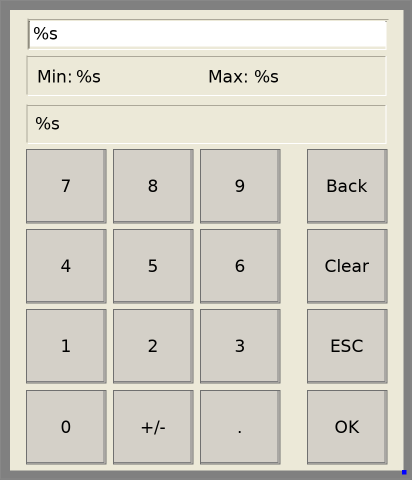
VISUALIZATION Custom_Numpad  // 412x480
VAR_INPUT
	stVariableValue : STRING;
	stMin : STRING;
	stMax : STRING;
	stTitle : STRING;
	flags : DWORD;
END_VAR
VAR
	bInit : BOOL;
	stMessage : STRING;
	stOutputValue : STRING;
END_VAR
    Rectangle (0,0 412x480)
    Rectangle (10,142 393x83)
    Rectangle (10,225 393x80)
    Rectangle (10,305 393x80)
    Rectangle (10,385 393x85)
    Button (307,390 80x74), "OK"
        OnMouseDown: CloseDialog Dialog=Custom_Numpad, Result=OK, NumpadKeypad=True, NumpadKeypadSet=True
    Button (307,309 80x74), "ESC"
        OnMouseDown: CloseDialog Dialog=Custom_Numpad, Result=Cancel, NumpadKeypad=True, NumpadKeypadSet=True
    Button (307,229 80x74), "Clear"
        OnMouseDown: execute {
            stVariableValue := '';
            stOutputValue := '';
            flags := flags AND 16#0008;
            flags := flags AND 16#0010;
        }
    Button (307,149 80x74), "Back"
        OnMouseDown: execute { VisuDlg_CheckedBack(stOutputValue, stVariableValue, bInit); }
    Button (200,390 80x74), "."
        OnMouseDown: execute { VisuDlg_CheckedAppend(stOutputValue, stVariableValue, bInit, (flags AND VisuElems.Visu_InputFlags.Password) = 1, '.'); }
    Button (113,390 80x74), "+/-"
        OnMouseDown: execute { VisuDlg_CheckedChangeSign(stOutputValue, stVariableValue, bInit, (flags AND VisuElems.Visu_InputFlags.Password) = 1); }
    Button (26,390 80x74), "0"
        OnMouseDown: execute { VisuDlg_CheckedAppend(stOutputValue, stVariableValue, bInit, (flags AND VisuElems.Visu_InputFlags.Password) = 1, '0'); }
    Button (26,309 80x74), "1"
        OnMouseDown: execute { VisuDlg_CheckedAppend(stOutputValue, stVariableValue, bInit, (flags AND VisuElems.Visu_InputFlags.Password) = 1, '1'); }
    Button (113,309 80x74), "2"
        OnMouseDown: execute { VisuDlg_CheckedAppend(stOutputValue, stVariableValue, bInit, (flags AND VisuElems.Visu_InputFlags.Password) = 1, '2'); }
    Button (200,309 80x74), "3"
        OnMouseDown: execute { VisuDlg_CheckedAppend(stOutputValue, stVariableValue, bInit, (flags AND VisuElems.Visu_InputFlags.Password) = 1, '3'); }
    Button (26,229 80x74), "4"
        OnMouseDown: execute { VisuDlg_CheckedAppend(stOutputValue, stVariableValue, bInit, (flags AND VisuElems.Visu_InputFlags.Password) = 1, '4'); }
    Button (113,229 80x74), "5"
        OnMouseDown: execute { VisuDlg_CheckedAppend(stOutputValue, stVariableValue, bInit, (flags AND VisuElems.Visu_InputFlags.Password) = 1, '5'); }
    Button (200,229 80x74), "6"
        OnMouseDown: execute { VisuDlg_CheckedAppend(stOutputValue, stVariableValue, bInit, (flags AND VisuElems.Visu_InputFlags.Password) = 1, '6'); }
    Button (26,149 80x74), "7"
        OnMouseDown: execute { VisuDlg_CheckedAppend(stOutputValue, stVariableValue, bInit, (flags AND VisuElems.Visu_InputFlags.Password) = 1, '7'); }
    Button (113,149 80x74), "8"
        OnMouseDown: execute { VisuDlg_CheckedAppend(stOutputValue, stVariableValue, bInit, (flags AND VisuElems.Visu_InputFlags.Password) = 1, '8'); }
    Button (200,149 80x74), "9"
        OnMouseDown: execute { VisuDlg_CheckedAppend(stOutputValue, stVariableValue, bInit, (flags AND VisuElems.Visu_InputFlags.Password) = 1, '9'); }
    Rectangle (10,10 393x48)
    Rectangle (10,57 393x85)
    Rectangle (73,64 127x25), "%s", text variable: stMin, invisible if: LEN(stMin) = 0
    Rectangle (251,64 127x25), "%s", text variable: stMax, invisible if: LEN(stMax) = 0
    Rectangle (205,64 45x25), "Max:", text variable: stMin, invisible if: LEN(stMax) = 0
        p55702900: SEL(((UDINT_TO_DINT(flags AND 16#0010))=16#0010),16#FF000000,16#FFFF0000)
    Rectangle (402,470 4x4)
    Polyline (27,94) (27,56) (385,56)
    Polyline (27,142) (27,105) (385,105)
    Polyline (28,49) (28,19) (388,19)
    Polyline (28,143) (386,143) (386,105)
    Polyline (28,95) (386,95) (386,56)
    Polyline (29,49) (386,49) (386,21)
    Polyline (29,48) (29,21) (386,21)
    Rectangle (32,111 349x25), "%s", text variable: stMessage
    Rectangle (34,64 41x25), "Min:", text variable: stMin, invisible if: LEN(stMin) = 0
        p55702900: SEL(((UDINT_TO_DINT(flags AND 16#0008))=16#0008),16#FF000000,16#FFFF0000)
    Rectangle (30,21 355x25), "%s", text variable: stOutputValue
    hotkey HotkeyInput Id=481049968640, Key=KeyDown=True, KeyName=0, ActionToExecute=Action=STSnippet=VisuDlg_CheckedAppend(stOutputValue, stVariableValue, bInit, (flags AND VisuElems.Visu_InputFlags.Password) = 1, '0');, VisuElemId=-1
    hotkey HotkeyInput Id=481053114368, Key=KeyDown=True, KeyName=NUM0, ActionToExecute=Action=STSnippet=VisuDlg_CheckedAppend(stOutputValue, stVariableValue, bInit, (flags AND VisuElems.Visu_InputFlags.Password) = 1, '0');, VisuElemId=-1
    hotkey HotkeyInput Id=481054162944, Key=KeyDown=True, KeyName=1, ActionToExecute=Action=STSnippet=VisuDlg_CheckedAppend(stOutputValue, stVariableValue, bInit, (flags AND VisuElems.Visu_InputFlags.Password) = 1, '1');, VisuElemId=-1
    hotkey HotkeyInput Id=481055211520, Key=KeyDown=True, KeyName=NUM1, ActionToExecute=Action=STSnippet=VisuDlg_CheckedAppend(stOutputValue, stVariableValue, bInit, (flags AND VisuElems.Visu_InputFlags.Password) = 1, '1');, VisuElemId=-1
    hotkey HotkeyInput Id=481056260096, Key=KeyDown=True, KeyName=2, ActionToExecute=Action=STSnippet=VisuDlg_CheckedAppend(stOutputValue, stVariableValue, bInit, (flags AND VisuElems.Visu_InputFlags.Password) = 1, '2');, VisuElemId=-1
    hotkey HotkeyInput Id=481057308672, Key=KeyDown=True, KeyName=NUM2, ActionToExecute=Action=STSnippet=VisuDlg_CheckedAppend(stOutputValue, stVariableValue, bInit, (flags AND VisuElems.Visu_InputFlags.Password) = 1, '2');, VisuElemId=-1
    hotkey HotkeyInput Id=481058357248, Key=KeyDown=True, KeyName=3, ActionToExecute=Action=STSnippet=VisuDlg_CheckedAppend(stOutputValue, stVariableValue, bInit, (flags AND VisuElems.Visu_InputFlags.Password) = 1, '3');, VisuElemId=-1
    hotkey HotkeyInput Id=481059405824, Key=KeyDown=True, KeyName=NUM3, ActionToExecute=Action=STSnippet=VisuDlg_CheckedAppend(stOutputValue, stVariableValue, bInit, (flags AND VisuElems.Visu_InputFlags.Password) = 1, '3');, VisuElemId=-1
    hotkey HotkeyInput Id=481060454400, Key=KeyDown=True, KeyName=4, ActionToExecute=Action=STSnippet=VisuDlg_CheckedAppend(stOutputValue, stVariableValue, bInit, (flags AND VisuElems.Visu_InputFlags.Password) = 1, '4');, VisuElemId=-1
    hotkey HotkeyInput Id=481061502976, Key=KeyDown=True, KeyName=NUM4, ActionToExecute=Action=STSnippet=VisuDlg_CheckedAppend(stOutputValue, stVariableValue, bInit, (flags AND VisuElems.Visu_InputFlags.Password) = 1, '4');, VisuElemId=-1
    hotkey HotkeyInput Id=481062551552, Key=KeyDown=True, KeyName=5, ActionToExecute=Action=STSnippet=VisuDlg_CheckedAppend(stOutputValue, stVariableValue, bInit, (flags AND VisuElems.Visu_InputFlags.Password) = 1, '5');, VisuElemId=-1
    hotkey HotkeyInput Id=481063600128, Key=KeyDown=True, KeyName=NUM5, ActionToExecute=Action=STSnippet=VisuDlg_CheckedAppend(stOutputValue, stVariableValue, bInit, (flags AND VisuElems.Visu_InputFlags.Password) = 1, '5');, VisuElemId=-1
    hotkey HotkeyInput Id=481064648704, Key=KeyDown=True, KeyName=6, ActionToExecute=Action=STSnippet=VisuDlg_CheckedAppend(stOutputValue, stVariableValue, bInit, (flags AND VisuElems.Visu_InputFlags.Password) = 1, '6');, VisuElemId=-1
    hotkey HotkeyInput Id=481065697280, Key=KeyDown=True, KeyName=NUM6, ActionToExecute=Action=STSnippet=VisuDlg_CheckedAppend(stOutputValue, stVariableValue, bInit, (flags AND VisuElems.Visu_InputFlags.Password) = 1, '6');, VisuElemId=-1
    hotkey HotkeyInput Id=481066745856, Key=KeyDown=True, KeyName=7, ActionToExecute=Action=STSnippet=VisuDlg_CheckedAppend(stOutputValue, stVariableValue, bInit, (flags AND VisuElems.Visu_InputFlags.Password) = 1, '7');, VisuElemId=-1
    hotkey HotkeyInput Id=481067794432, Key=KeyDown=True, KeyName=NUM7, ActionToExecute=Action=STSnippet=VisuDlg_CheckedAppend(stOutputValue, stVariableValue, bInit, (flags AND VisuElems.Visu_InputFlags.Password) = 1, '7');, VisuElemId=-1
    hotkey HotkeyInput Id=481068843008, Key=KeyDown=True, KeyName=8, ActionToExecute=Action=STSnippet=VisuDlg_CheckedAppend(stOutputValue, stVariableValue, bInit, (flags AND VisuElems.Visu_InputFlags.Password) = 1, '8');, VisuElemId=-1
    hotkey HotkeyInput Id=481069891584, Key=KeyDown=True, KeyName=NUM8, ActionToExecute=Action=STSnippet=VisuDlg_CheckedAppend(stOutputValue, stVariableValue, bInit, (flags AND VisuElems.Visu_InputFlags.Password) = 1, '8');, VisuElemId=-1
    hotkey HotkeyInput Id=481070940160, Key=KeyDown=True, KeyName=9, ActionToExecute=Action=STSnippet=VisuDlg_CheckedAppend(stOutputValue, stVariableValue, bInit, (flags AND VisuElems.Visu_InputFlags.Password) = 1, '9');, VisuElemId=-1
    hotkey HotkeyInput Id=481071988736, Key=KeyDown=True, KeyName=NUM9, ActionToExecute=Action=STSnippet=VisuDlg_CheckedAppend(stOutputValue, stVariableValue, bInit, (flags AND VisuElems.Visu_InputFlags.Password) = 1, '9');, VisuElemId=-1
    hotkey HotkeyInput Id=481073037312, Key=KeyDown=True, KeyName=SUBTRACT, ActionToExecute=Action=STSnippet=VisuDlg_CheckedChangeSign(stOutputValue, stVariableValue, bInit, (flags AND VisuElems.Visu_InputFlags.Password) = 1);, VisuElemId=-1
    hotkey HotkeyInput Id=481074085888, Key=KeyDown=True, KeyName=COMMA, ActionToExecute=Action=STSnippet=VisuDlg_CheckedAppend(stOutputValue, stVariableValue, bInit, (flags AND VisuElems.Visu_InputFlags.Password) = 1, '.');, VisuElemId=-1
    hotkey HotkeyInput Id=481075134464, Key=KeyDown=True, KeyName=BACKSPACE, ActionToExecute=Action=STSnippet=VisuDlg_CheckedBack(stOutputValue, stVariableValue, bInit);, VisuElemId=-1
    hotkey HotkeyInput Id=481076183040, Key=KeyDown=True, KeyName=DELETE, ActionToExecute=Action=STSnippet=stVariableValue := ''; stOutputValue := ''; flags := flags AND 16#0008; flags := flags AND 16#0010;, VisuElemId=-1
    hotkey HotkeyInput Id=481077231616, Key=KeyDown=True, KeyName=ESCAPE, ActionToExecute=Action=Dialog=Custom_Numpad, Result=Cancel, NumpadKeypad=True, NumpadKeypadSet=True, VisuElemId=-1
    hotkey HotkeyInput Id=481078280192, Key=KeyDown=True, KeyName=RETURN_KEY, ActionToExecute=Action=Dialog=Custom_Numpad, Result=OK, NumpadKeypad=True, NumpadKeypadSet=True, VisuElemId=-1
END_VISUALIZATION

(* stored: Version 1.1.0.1, ProductVersion 3.1.4024.3
   Visu Custom_Numpad: Id {1ba8af01-78cb-464b-a67e-a242742044ce} *)
